// TIA Portal V20 export
DATA_BLOCK "DB_Recipe"   // DB133
// stored: InstanceOfName FB_Recipe, InstanceOfType FB
"FB_Recipe"
BEGIN
END_DATA_BLOCK
